{attribute 'qualified_only'}
{attribute 'strict'}
TYPE E_Checkvalvereject :
(
	enum_member         := 0,
    CheckvalveOk        := 10,
    Checkvalvefailure   := 20
);
END_TYPE

(* stored: Version 1.1.0.1, ProductVersion 3.1.4024.12
   DUT E_Checkvalvereject: Id {98fbf3a4-345c-4e23-a337-224819a5a35e} *)
